	            IF ("IdbC05_Loader".M_01.startedForward OR NOT "DbDeviceONOF".boolValues[4])
	                AND ("IdbC05_Loader".M_02.startedForward OR NOT "DbDeviceONOF".boolValues[5])
	                AND (NOT "IdbC05_Loader".M_03.startedForward OR NOT "DbDeviceONOF".boolValues[6])
	                AND (NOT "IdbC05_Loader".M_04.startedForward OR NOT "DbDeviceONOF".boolValues[7])
	                OR #HMINexStep THEN
	                #HMINexStep := FALSE;
	                #StepOld := #Step;
	                #TimeCurrentStep := 0;
	                #Step := 34;

	            ELSIF #HMIStopProg THEN // Переход на сушильную продувку
	                #StepOld := #Step;
	                #TimeCurrentStep := 0;
	                #Step := 50;

	            ELSIF #HMIStop THEN // Переход на стоповый шаг
	                #HMIStop := 0;
	                #StepOld := #Step;
	                #TimeCurrentStep := 0;
	                #Step := 80;
	            END_IF;

	        34: //Сушка. Выход на заданную температуру
	            #TimeCurrentStep := #TimeCurrentStep + #cycleTime; //Подсчет времени текущей программы

	            //Передача параметров регулирования и старт горелок до момента подтверждения оператором остановки
	            "DbRegulatorsRetain".instMe[0].setpoint := "DbRegulatorsRetain".instMe[1].setpoint :=
	            "DbU1_Recipe".TemSet_2;

	            "DbRegulatorsRetain".instMe[0].hysteresys.stage_1 := "DbRegulatorsRetain".instMe[1].hysteresys.stage_1 :=
	            "DbU1_Recipe".GistHigh_2;

	            "DbRegulatorsRetain".instMe[0].hysteresys.stage_2 := "DbRegulatorsRetain".instMe[1].hysteresys.stage_2 :=
	            "DbU1_Recipe".GistLow_2;

	            #TimetUsed(START := TRUE,
	                       NUM := 4,
	                       TIM := 1800,
	                       SAMPLE_T := #cycleTime);

	            IF (#TemSet_2 - 2) <= ("IdbC03_Loader".TT7_10.value) OR #HMINexStep THEN
	                #HMINexStep := FALSE;
	                #StepOld := #Step;
	                #TimeCurrentStep := 0;
	                #Step := 35;
	                #TimetUsed(START := FALSE,
	                           NUM := 4);

	            ELSIF #HMIStopProg THEN // Переход на сушильную продувку
	                #StepOld := #Step;
	                #TimeCurrentStep := 0;
	                #Step := 50;

	            ELSIF #HMIStop THEN // Переход на стоповый шаг
	                #HMIStop := 0;
	                #StepOld := #Step;
	                #TimeCurrentStep := 0;
	                #Step := 80;
	            END_IF;

	        35: //Сушка. Отсчет заданного времени
	            #TimeCurrentStep := #TimeCurrentStep + #cycleTime; //Подсчет времени текущей программы
	            #TimeDryingRun := #TimeDryingRun + #cycleTime;

	            IF #TimeDryingRun > #TimeDryingSet OR #HMINexStep THEN
	                #HMINexStep := FALSE;
	                #StepOld := #Step;
	                #TimeCurrentStep := 0;
	                #Step := 50;

	            ELSIF #HMIStop THEN // Переход на стоповый шаг
	                #HMIStop := 0;
	                #StepOld := #Step;
	                #TimeCurrentStep := 0;
	                #Step := 80;

	            ELSIF #HMIStopProg THEN // Переход на сушильную продувку по кнопке
	                #StepOld := #Step;
	                #TimeCurrentStep := 0;
	                #Step := 50;

	          //  ELSIF #HMIStartClor THEN // Переход на Покраску по кнопке
	          //     #StepOld := #Step;
	          //      #TimeCurrentStep := 0;
	          //      #Step := 10;
	            END_IF;

	        40: //Окрасочная продувка
	            //Жалюзи Y1-2 открыты, приточный и вытяжные вентиляторы запущены, горелки работают.
	            //Условиями отключения режима являются: падение температуры до заданной в рецепте (условно +20)
	            //При выполнении условия продувка работает ещё около 3 минут и отключается.
	            #TimeCurrentStep := #TimeCurrentStep + #cycleTime; //Подсчет времени текущей программы

	            // Активация  и проверка положения клапанов  как для покраски
	            IF ("IdbC06_Loader".Y_1.activated OR NOT "DbDeviceONOF".boolValues[10])
	                AND ("IdbC06_Loader".Y_2.activated OR NOT "DbDeviceONOF".boolValues[11])
	                OR #HMINexStep THEN
	                #HMINexStep := FALSE;
	                #StepOld := #Step;
	                #Step := 41;

	            ELSIF #HMIStopProg THEN // Переход на стоповый шаг
	                #StepOld := #Step;
	                #TimeCurrentStep := 0;
	                #Step := 80;

	            ELSIF #HMIStop THEN // Переход на стоповый шаг
	                #HMIStop := 0;
	                #StepOld := #Step;
	                #TimeCurrentStep := 0;
	                #Step := 80;
	            END_IF;

	        41: // Окрасочная продувка: Активация приточных и вытяжных вентиляторов
	            #TimeCurrentStep := #TimeCurrentStep + #cycleTime; //Подсчет времени текущей программы

	            IF (("IdbC05_Loader".M_01.startedForward OR NOT "DbDeviceONOF".boolValues[4])
	                AND ("IdbC05_Loader".M_02.startedForward OR NOT "DbDeviceONOF".boolValues[5])
	                AND ("IdbC05_Loader".M_03.startedForward OR NOT "DbDeviceONOF".boolValues[6])
	                AND ("IdbC05_Loader".M_04.startedForward OR NOT "DbDeviceONOF".boolValues[7]))
	                OR #HMINexStep THEN
	                #HMINexStep := FALSE;
	                #StepOld := #Step;
	                #Step := 42;

	            ELSIF #HMIStopProg THEN // Переход на стоповый шаг
	                #StepOld := #Step;
	                #TimeCurrentStep := 0;
	                #Step := 80;

	            ELSIF #HMIStop THEN // Переход на стоповый шаг
	                #HMIStop := 0;
	                #StepOld := #Step;
	                #TimeCurrentStep := 0;
	                #Step := 80;
	            END_IF;

	        42: //Окрасочная продувка : Охлаждение до заданной температуры
	            #TimeCurrentStep := #TimeCurrentStep + #cycleTime; //Подсчет времени текущей программы
	            #TimePurgeRun := #TimePurgeRun + #cycleTime;

	            // Подсчет времени продувки и проверка температуры
	            // При достижение темературы до уставки, а так же при превышении максимального времени переход
	            IF #TimetUsed.done_arr[3] OR #TimePurgeRun >= #TimePurgSet
	                OR #HMINexStep THEN
	                #HMINexStep := FALSE;
	                #StepOld := #Step;
	                #Step := 80;

	            ELSIF #HMIStopProg THEN // Переход на стоповый шаг
	                #StepOld := #Step;
	                #TimeCurrentStep := 0;
	                #Step := 80;

	            ELSIF #HMIStop THEN // Переход на стоповый шаг
	                #HMIStop := 0;
	                #StepOld := #Step;
	                #TimeCurrentStep := 0;
	                #Step := 80;

	            ELSIF "DbU1_Recipe".TemSet_3 + 2 >= "IdbC03_Loader".TT7_10.value THEN
	                #TimetUsed(START := TRUE,
	                           NUM := 3,
	                           TIM := 180,
	                           SAMPLE_T := #cycleTime);
	            END_IF;

	        50:  // Сушильная продувка
	            #TimeCurrentStep := #TimeCurrentStep + #cycleTime; //Подсчет времени текущей программы

	            // Активация и проверка положения клапанов как для сушки
	            IF "IdbC06_Loader".Y_1.deactivated AND "IdbC06_Loader".Y_2.deactivated
	                OR #HMINexStep THEN
	                #HMINexStep := FALSE;
	                #StepOld := #Step;
	                #Step := 52;

	            ELSIF #HMIStopProg THEN // Переход на стоповый шаг
	                #StepOld := #Step;
	                #TimeCurrentStep := 0;
	                #Step := 80;

	            ELSIF #HMIStop THEN // Переход на стоповый шаг
	                #HMIStop := 0;
	                #StepOld := #Step;
	                #TimeCurrentStep := 0;
	                #Step := 80;
	            END_IF;

	        52: //Сушильная продувка. Ожидание снижения температуры.
	            #TimeCurrentStep := #TimeCurrentStep + #cycleTime; //Подсчет времени текущей программы
	            #TimePurgeRun := #TimePurgeRun + #cycleTime;

	            IF #TimetUsed.done_arr[3] OR #TimePurgeRun >= #TimePurgSet
	                OR #HMINexStep THEN
	                #HMINexStep := FALSE;
	                #StepOld := #Step;
	                #Step := 80;

	            ELSIF #HMIStopProg THEN // Переход на стоповый шаг
	                #StepOld := #Step;
	                #TimeCurrentStep := 0;
	                #Step := 80;

	            ELSIF #HMIStop THEN // Переход на стоповый шаг
	                #HMIStop := 0;
	                #StepOld := #Step;
	                #TimeCurrentStep := 0;
	                #Step := 80;

	            ELSIF "DbU1_Recipe".TemSet_3 + 2 >= "IdbC03_Loader".TT7_10.value THEN
	                #TimetUsed(START := TRUE,
	                           NUM := 3,
	                           TIM := 180,
	                           SAMPLE_T := #cycleTime);
	            END_IF;

	        80: // Штатная остановка ожидание завершение работы двигателей
	            #TimeCurrentStep := #TimeCurrentStep + #cycleTime; //Подсчет времени текущей программы

	            // Сброс параметров регулятора
	            "DbRegulatorsRetain".instMe[0].setpoint := "DbRegulatorsRetain".instMe[1].setpoint := 0.0;

	            "DbRegulatorsRetain".instMe[0].hysteresys.stage_1 := "DbRegulatorsRetain".instMe[1].hysteresys.stage_1 := 0.0;

	            "DbRegulatorsRetain".instMe[0].hysteresys.stage_2 := "DbRegulatorsRetain".instMe[1].hysteresys.stage_2 := 0.0;

	            //Проверка положения задвижек на соответствие завершающему шагу
	            IF NOT "IdbC06_Loader".Y_1.activated AND NOT "IdbC06_Loader".Y_2.activated
	                OR #HMINexStep THEN
	                #HMIStopProg := FALSE;
	                #HMINexStep := FALSE;
	                #StepOld := #Step;
	                #Step := 81;
	            END_IF;

	        81: // Штатная остановка ожидание завершение работы двигателей
	            #TimeCurrentStep := #TimeCurrentStep + #cycleTime; //Подсчет времени текущей программы

	            IF #TimeCurrentStep > 1
	                OR #HMINexStep THEN
	                #HMIStop := FALSE;
	                #HMINexStep := FALSE;
	                #StepOld := #Step;
	                #Step := 0;
	                #TimeCurrentStep := 0;
	            END_IF;

	        91: // Авария. Нажата аварийная кнопка
	            #TimeCurrentStep := #TimeCurrentStep + #cycleTime; //Подсчет времени текущей программы

	            IF #resetErrorCode  // Если нет этой аварии и нажата кнопка сброс, переходим на начальный шаг
	                AND   NOT #StorErr THEN
	                #StepOld := #Step;
	                #Step := 80;
	                #TimeCurrentStep := 0;
	            END_IF;

	        92: // Авария. Пожар
	            #TimeCurrentStep := #TimeCurrentStep + #cycleTime; //Подсчет времени текущей программы

	            IF #resetErrorCode  // Если нет этой аварии и нажата кнопка сброс, переходим на начальный шаг
	                AND NOT #FirerErr THEN
	                #StepOld := #Step;
	                #Step := 80;
	                #TimeCurrentStep := 0;
	            END_IF;

	        94: // Авария. Электропривода вентиляторов
	            #TimeCurrentStep := #TimeCurrentStep + #cycleTime; //Подсчет времени текущей программы

	            IF #resetErrorCode  // Если нет этой аварии и нажата кнопка сброс, переходим на начальный шаг
	                AND NOT #tempMotorError THEN
	                #StepOld := #Step;
	                #Step := 80;
	                #TimeCurrentStep := 0;

	            ELSIF #HMIStopProg THEN // Переход на стоповый шаг
	                #StepOld := #Step;
	                #TimeCurrentStep := 0;
	                #Step := 80;

	            ELSIF #HMIStop THEN // Переход на стоповый шаг
	                #StepOld := #Step;
	                #TimeCurrentStep := 0;
	                #Step := 80;

	            ELSIF #TimetUsed.done_arr[3] OR #TimePurgeRun >= #TimePurgSet THEN
	                #HMINexStep := FALSE;
	                #StepOld := #Step;
	                #Step := 80;

	            ELSIF "DbU1_Recipe".TemSet_3 + 2 >= "IdbC03_Loader".TT7_10.value THEN
	                #TimetUsed(START := TRUE,
	                           NUM := 3,
	                           TIM := 180,
	                           SAMPLE_T := #cycleTime);
	            END_IF;

	        95: // Авария. Высокая температура в камере.
	            #TimeCurrentStep := #TimeCurrentStep + #cycleTime; //Подсчет времени текущей программы

	            IF #resetErrorCode  // Если нет этой аварии и нажата кнопка сброс, переходим на начальный шаг
	                AND NOT #tempHiTempErr THEN
	                #StepOld := #Step;
	                #Step := 80;
	                #TimeCurrentStep := 0;

	            ELSIF #HMIStopProg THEN // Переход на стоповый шаг
	                #StepOld := #Step;
	                #TimeCurrentStep := 0;
	                #Step := 80;

	            ELSIF #HMIStop THEN // Переход на стоповый шаг
	                #StepOld := #Step;
	                #TimeCurrentStep := 0;
	                #Step := 80;

	            ELSIF #TimetUsed.done_arr[3] OR #TimePurgeRun >= #TimePurgSet THEN
	                #HMINexStep := FALSE;
	                #StepOld := #Step;
	                #Step := 80;

	            ELSIF "DbU1_Recipe".TemSet_3 + 2 >= "IdbC03_Loader".TT7_10.value THEN
	                #TimetUsed(START := TRUE,
	                           NUM := 3,
	                           TIM := 180,
	                           SAMPLE_T := #cycleTime);
	            END_IF;

	        96: // Авария. Авария оборудования.
	            #TimeCurrentStep := #TimeCurrentStep + #cycleTime; //Подсчет времени текущей программы

	            // Сброс параметров регулятора
	            "DbRegulatorsRetain".instMe[0].setpoint := "DbRegulatorsRetain".instMe[1].setpoint := 0.0;

	            "DbRegulatorsRetain".instMe[0].hysteresys.stage_1 := "DbRegulatorsRetain".instMe[1].hysteresys.stage_1 := 0.0;

	            "DbRegulatorsRetain".instMe[0].hysteresys.stage_2 := "DbRegulatorsRetain".instMe[1].hysteresys.stage_2 := 0.0;

	            IF #resetErrorCode  // Если нет этой аварии и нажата кнопка сброс, переходим на начальный шаг
	                AND NOT #tempEquipmentError THEN
	                #StepOld := #Step;
	                #Step := 80;
	                #TimeCurrentStep := 0;

	            ELSIF #HMIStopProg THEN // Переход на стоповый шаг
	                #StepOld := #Step;
	                #TimeCurrentStep := 0;
	                #Step := 80;

	            ELSIF #HMIStop THEN // Переход на стоповый шаг
	                #StepOld := #Step;
	                #TimeCurrentStep := 0;
	                #Step := 80;

	            ELSIF #TimetUsed.done_arr[3] OR #TimePurgeRun >= #TimePurgSet THEN
	                #HMINexStep := FALSE;
	                #StepOld := #Step;
	                #Step := 80;

	            ELSIF "DbU1_Recipe".TemSet_3 + 2 >= "IdbC03_Loader".TT7_10.value THEN
	                #TimetUsed(START := TRUE,
	                           NUM := 3,
	                           TIM := 180,
	                           SAMPLE_T := #cycleTime);
	            END_IF;

	        97: // Авария. Сторожевой таймер.
	            #TimeCurrentStep := #TimeCurrentStep + #cycleTime; //Подсчет времени текущей программы

	            IF #resetErrorCode  // Если нет этой аварии и нажата кнопка сброс, переходим на начальный шаг
	                AND NOT #tempWatchdogErr THEN
	                #TimeCurrentStep := 0;
	                #StepOld := #Step;
	                #Step := 80;

	            ELSIF #HMIStopProg THEN // Переход на стоповый шаг
	                #StepOld := #Step;
	                #TimeCurrentStep := 0;
	                #Step := 80;

	            ELSIF #HMIStop THEN // Переход на стоповый шаг
	                #StepOld := #Step;
	                #TimeCurrentStep := 0;
	                #Step := 80;
	            END_IF;
	    END_CASE;
	END_REGION

	REGION Активация устройств

	    CASE #Step OF

	        10, 40: // Активация начального положения задвижек. Для программы окраски
	                // задвижки Y1-2 открыты
	            IF "DbDeviceONOF".boolValues[10] THEN
	                    "IdbC06_Loader".Y_1.autoDeactivate := FALSE;
	                    "IdbC06_Loader".Y_1.autoActivate := TRUE;
	                END_IF;
	                IF "DbDeviceONOF".boolValues[11] THEN
	                    "IdbC06_Loader".Y_2.autoDeactivate := FALSE;
	                    "IdbC06_Loader".Y_2.autoActivate := TRUE;
	                END_IF;

	            11, 41: //Поочередная активация двигателей для покраски
	                //Поочередная активация двигателей
	            CASE #EM.group OF
	                #EMPTY:
	                    #EM.group := #M1_START_RELEASE;
	                    IF #TimetUsed.done_arr[1] THEN
	                        #TimetUsed(START := TRUE,
	                                   NUM := 1,
	                                   TIM := #TimeOnMotor,
	                                   SAMPLE_T := #cycleTime);
	                    END_IF;

	                    //Активация востребованности двигателей через задержку по времени
	                #M1_START_RELEASE:
	                    #TimetUsed(START := TRUE,
	                               NUM := 1,
	                               TIM := #TimeOnMotor,
	                               SAMPLE_T := #cycleTime);
	                    IF #TimetUsed.done_arr[1] THEN
	                        #EM.group := #M3_START_RELEASE;
	                        #TimetUsed(START := FALSE,
	                                   NUM := 1);
	                    END_IF;

	                #M3_START_RELEASE:
	                    #TimetUsed(START := TRUE,
	                               NUM := 1,
	                               TIM := #TimeOnMotor,
	                               SAMPLE_T := #cycleTime);
	                    IF #TimetUsed.done_arr[1] THEN
	                        #EM.group := #M2_START_RELEASE;
	                        #TimetUsed(START := FALSE,
	                                   NUM := 1);
	                    END_IF;

	                #M2_START_RELEASE:
	                    #TimetUsed(START := TRUE,
	                               NUM := 1,
	                               TIM := #TimeOnMotor,
	                               SAMPLE_T := #cycleTime);
	                    IF #TimetUsed.done_arr[1] THEN
	                        #EM.group := #M4_START_RELEASE;
	                        #TimetUsed(START := FALSE,
	                                   NUM := 1);
	                    END_IF;

	                #M4_START_RELEASE:
	                    #EM.group := #DONE;

	                #DONE:
	                    #TimetUsed(START := TRUE,
	                               NUM := 1,
	                               TIM := #TimeOnMotor,
	                               SAMPLE_T := #cycleTime);
	                    IF #TimetUsed.done_arr[1] THEN
	                        #TimetUsed(START := FALSE,
	                                   NUM := 1);
	                        #EM.group := #EMPTY;
	                    END_IF;
	                ELSE
	                    #EM.group := #EMPTY;
	                    #TimetUsed(START := FALSE,
	                               NUM := 1);
	            END_CASE;

	            // Непосредственное включение двигателей при их востребованности и разрешение (активен бит их участия в работе HMI)
	            IF ("DbDeviceONOF".boolValues[4] AND ((#EM.group >= #M1_START_RELEASE))) THEN
	                "IdbC05_Loader".M_01.autoStartForward := TRUE;
	            END_IF;
	            IF "DbDeviceONOF".boolValues[5] AND (#EM.group >= #M2_START_RELEASE) THEN
	                "IdbC05_Loader".M_02.autoStartForward := TRUE;
	            END_IF;
	            IF ("DbDeviceONOF".boolValues[6] AND (#EM.group >= #M3_START_RELEASE)) THEN
	                "IdbC05_Loader".M_03.autoStartForward := TRUE;
	            END_IF;
	            IF ("DbDeviceONOF".boolValues[7] AND (#EM.group >= #M4_START_RELEASE)) THEN
	                "IdbC05_Loader".M_04.autoStartForward := TRUE;
	            END_IF;

	        12: //Непосредственное включение двигателей и горелок для покраски.
	            //Активация горелок
	            IF "DbDeviceONOF".boolValues[8] THEN
	                "IdbC08_Loader".Regul_1.release := TRUE;
	            END_IF;
	            IF "DbDeviceONOF".boolValues[9] THEN
	                "IdbC08_Loader".Regul_2.release := TRUE;
	            END_IF;

	        30: //Переключение клапанов в режим сушки Y1-2 закрываются
	            //Активация горелок в случае деактивации. Двигатели продолжают работы до перехода на следующий шаг
	            //Деактивация горелок
	            IF "DbDeviceONOF".boolValues[8] THEN
	                "IdbC08_Loader".Regul_1.release := FALSE;
	            END_IF;
	            IF "DbDeviceONOF".boolValues[9] THEN
	                "IdbC08_Loader".Regul_2.release := FALSE;
	            END_IF;

	            // Деактивация двигателей
	            "IdbC05_Loader".M_01.autoStartForward := "IdbC05_Loader".M_02.autoStartForward := "IdbC05_Loader".M_03.autoStartForward := "IdbC05_Loader".M_04.autoStartForward := FALSE;

	            //Переключение клапанов в режим сушки
	            IF "DbDeviceONOF".boolValues[10] THEN
	                "IdbC06_Loader".Y_1.autoActivate := FALSE;
	                "IdbC06_Loader".Y_1.autoDeactivate := TRUE;
	            END_IF;
	            IF "DbDeviceONOF".boolValues[11] THEN
	                "IdbC06_Loader".Y_2.autoActivate := FALSE;
	                "IdbC06_Loader".Y_2.autoDeactivate := TRUE;
	            END_IF;

	        32:  // Поочередное включение двигателей
	                CASE #EM.group OF
	                    #EMPTY:
	                        #EM.group := #M1_START_RELEASE;
	                        IF #TimetUsed.done_arr[1] THEN
	                            #TimetUsed(START := TRUE,
	                                       NUM := 1,
	                                       TIM := #TimeOnMotor,
	                                       SAMPLE_T := #cycleTime);
	                        END_IF;

	                        //Активация востребованности двигателей через задержку по времени
	                    #M1_START_RELEASE:
	                        #TimetUsed(START := TRUE,
	                                   NUM := 1,
	                                   TIM := #TimeOnMotor,
	                                   SAMPLE_T := #cycleTime);
	                        IF #TimetUsed.done_arr[1] THEN
	                            #EM.group := #M2_START_RELEASE;
	                            #TimetUsed(START := FALSE,
	                                       NUM := 1);
	                        END_IF;

	                    #M2_START_RELEASE:
	                        #EM.group := #DONE;

	                    #DONE:
	                        #TimetUsed(START := TRUE,
	                                   NUM := 1,
	                                   TIM := #TimeOnMotor,
	                                   SAMPLE_T := #cycleTime);
	                        IF #TimetUsed.done_arr[1] THEN
	                            #EM.group := #EMPTY;
	                            #TimetUsed(START := FALSE,
	                                       NUM := 1);
	                        END_IF;
	                    ELSE
	                        #EM.group := #EMPTY;
	                        #TimetUsed(START := FALSE,
	                                   NUM := 1);
	                END_CASE;

	                // Непосредственное включение двигателей при их востребованности и разрешение (активен бит их участия в работе HMI)
	                IF ("DbDeviceONOF".boolValues[4] AND ((#EM.group >= #M1_START_RELEASE))) THEN
	                    "IdbC05_Loader".M_01.autoStartForward := TRUE;
	                END_IF;
	                IF "DbDeviceONOF".boolValues[5] AND (#EM.group >= #M2_START_RELEASE) THEN
	                    "IdbC05_Loader".M_02.autoStartForward := TRUE;
	                END_IF;
	                IF "DbDeviceONOF".boolValues[6] THEN
	                    "IdbC05_Loader".M_03.autoStartForward := FALSE;
	                END_IF;
	                IF "DbDeviceONOF".boolValues[7] THEN
	                    "IdbC05_Loader".M_04.autoStartForward := FALSE;
	                END_IF;

	        34: // Активация горелок
	            IF "DbDeviceONOF".boolValues[8] THEN
	                "IdbC08_Loader".Regul_1.release := TRUE;
	            END_IF;
	            IF "DbDeviceONOF".boolValues[9] THEN
	                "IdbC08_Loader".Regul_2.release := TRUE;
	            END_IF;

	        42: //Окрасочная продувка. Ожидание достижения уставок по времени или температуре
	            //Деактивация горелок
	            IF "DbDeviceONOF".boolValues[8] THEN
	                "IdbC08_Loader".Regul_1.release := FALSE;
	            END_IF;
	            IF "DbDeviceONOF".boolValues[9] THEN
	                "IdbC08_Loader".Regul_2.release := FALSE;
	            END_IF;

	        50: //Сушильная продувка
	            //Клапаны в режиме сушки, остаются в предыдущем положении
	            IF "DbDeviceONOF".boolValues[10] THEN
	                "IdbC06_Loader".Y_1.autoActivate := FALSE;
	                "IdbC06_Loader".Y_1.autoDeactivate := TRUE;
	            END_IF;
	            IF "DbDeviceONOF".boolValues[11] THEN
	                "IdbC06_Loader".Y_2.autoActivate := FALSE;
	                "IdbC06_Loader".Y_2.autoDeactivate := TRUE;
	            END_IF;

	        52: //Сушильная продувка
	            // Приточне двигатели продолжают работу, вытяжные деактивированы.
	            IF ("DbDeviceONOF".boolValues[4]) THEN
	                "IdbC05_Loader".M_01.autoStartForward := TRUE;
	            END_IF;
	            IF "DbDeviceONOF".boolValues[5] THEN
	                "IdbC05_Loader".M_02.autoStartForward := TRUE;
	            END_IF;
	            IF ("DbDeviceONOF".boolValues[6]) THEN
	                "IdbC05_Loader".M_03.autoStartForward := FALSE;
	            END_IF;
	            IF ("DbDeviceONOF".boolValues[7]) THEN
	                "IdbC05_Loader".M_04.autoStartForward := FALSE;
	            END_IF;

	            // Деактивация регулирования горелок
	            "IdbC08_Loader".Regul_1.release := FALSE;
	            "IdbC08_Loader".Regul_2.release := FALSE;

	        80:  //Переключенеи задвижек в первоначальное положение, дективация остального
	            // задвижек жалюзи Y1-2 закрыты
	            IF "DbDeviceONOF".boolValues[10] THEN
	                "IdbC06_Loader".Y_1.autoActivate := FALSE;
	                "IdbC06_Loader".Y_1.autoDeactivate := TRUE;
	            END_IF;
	            IF "DbDeviceONOF".boolValues[11] THEN
	                "IdbC06_Loader".Y_2.autoActivate := FALSE;
	                "IdbC06_Loader".Y_2.autoDeactivate := TRUE;
	            END_IF;

	            // Деактивация горелок
	            "IdbC08_Loader".Regul_1.release := FALSE;
	            "IdbC08_Loader".Regul_2.release := FALSE;

	            // Деактивация двигателей
	            "IdbC05_Loader".M_01.autoStartForward := "IdbC05_Loader".M_02.autoStartForward := "IdbC05_Loader".M_03.autoStartForward := "IdbC05_Loader".M_04.autoStartForward := FALSE;

	        81: // Деактивация всего
	            //Переключение камер задвижек 1-2
	            "IdbC06_Loader".Y_1.autoActivate := "IdbC06_Loader".Y_2.autoActivate := FALSE;
	            "IdbC06_Loader".Y_1.autoDeactivate := "IdbC06_Loader".Y_2.autoDeactivate := TRUE;

	            // Деактивация горелок
	            "IdbC08_Loader".Regul_1.release := FALSE;
	            "IdbC08_Loader".Regul_2.release := FALSE;

	            // Деактивация двигателей
	            "IdbC05_Loader".M_01.autoStartForward := "IdbC05_Loader".M_02.autoStartForward := "IdbC05_Loader".M_03.autoStartForward := "IdbC05_Loader".M_04.autoStartForward := FALSE;

	        91: //Нажата аварийная кнопка. Все отключить
	            // Аварийный останов активируетя до перехода на шаг
	            //Отключение в авто режиме
	            //Отключение   задвижек 1-2
	            "IdbC06_Loader".Y_1.autoActivate := "IdbC06_Loader".Y_2.autoActivate := FALSE;
	            "IdbC06_Loader".Y_1.autoDeactivate := "IdbC06_Loader".Y_2.autoDeactivate := TRUE;

	            // Деактивация горелок
	            "IdbC08_Loader".Regul_1.release := FALSE;
	            "IdbC08_Loader".Regul_2.release := FALSE;

	            // Деактивация двигателей
	            "IdbC05_Loader".M_01.autoStartForward := "IdbC05_Loader".M_02.autoStartForward := "IdbC05_Loader".M_03.autoStartForward := "IdbC05_Loader".M_04.autoStartForward := FALSE;

	        92: // Сигнал о пожаре. Y1-2 закрываются, свет горит на протяжении 30 секунд и отключается.
	            // Аварийный останов активируетя до перехода на шаг
	            //Отключение в авто режиме

	            //Переключение клапанов в режим сушки
	            IF "DbDeviceONOF".boolValues[10] THEN
	                "IdbC06_Loader".Y_1.autoActivate := FALSE;
	                "IdbC06_Loader".Y_1.autoDeactivate := TRUE;
	            END_IF;
	            IF "DbDeviceONOF".boolValues[11] THEN
	                "IdbC06_Loader".Y_2.autoActivate := FALSE;
	                "IdbC06_Loader".Y_2.autoDeactivate := TRUE;
	            END_IF;

	            "IdbC08_Loader".Regul_1.release := FALSE;
	            "IdbC08_Loader".Regul_2.release := FALSE;

	            // Деактивация двигателей
	            "IdbC05_Loader".M_01.autoStartForward := "IdbC05_Loader".M_02.autoStartForward := "IdbC05_Loader".M_03.autoStartForward := "IdbC05_Loader".M_04.autoStartForward := FALSE;

	        94: // Авария привода вентилятора
	            //Запускается режим продувки. Тип продувки зависит от того на какой из программ это произошло.
	            // Задвижки остаются в предыдущем положении

	            //Горелки останавливаются
	            "IdbC08_Loader".Regul_1.release := FALSE;
	            "IdbC08_Loader".Regul_2.release := FALSE;

	            // Активируются только приточка Если какой-то в аварии он и так не запустится
	            IF (#StepOld >= 30 AND #StepOld < 40) OR (#StepOld >= 50 AND #StepOld < 60) THEN // Если пред шаг связан с сушкой, то запускается сушильная продувка
	                "IdbC05_Loader".M_01.autoStartForward := "IdbC05_Loader".M_02.autoStartForward := TRUE;
	                "IdbC05_Loader".M_03.autoStartForward := "IdbC05_Loader".M_04.autoStartForward := FALSE;
	            ELSE // Иначе запускается продувка с работой всех двигателей
	                "IdbC05_Loader".M_01.autoStartForward := "IdbC05_Loader".M_02.autoStartForward := "IdbC05_Loader".M_03.autoStartForward := "IdbC05_Loader".M_04.autoStartForward := TRUE;
	            END_IF;

	        95, 96: // Авария  оборудования или Высокая температура в камере.
	            //Запускается режим продувки. Тип продувки зависит от того на какой из программ это произошло.
	            // Задвижки остаются в предыдущем положении
	            //Горелки останавливаются
	            "IdbC08_Loader".Regul_1.release := FALSE;
	            "IdbC08_Loader".Regul_2.release := FALSE;

	            // Активируются все двигатели. Если какой-то в аварии он и так не запустится
	            IF (#StepOld >= 30 AND #StepOld < 40) OR (#StepOld >= 50 AND #StepOld < 60) THEN // Если пред шаг связан с сушкой, то запускается сушильная продувка
	                "IdbC05_Loader".M_01.autoStartForward := "IdbC05_Loader".M_02.autoStartForward := TRUE;
	                "IdbC05_Loader".M_03.autoStartForward := "IdbC05_Loader".M_04.autoStartForward := FALSE;
	            ELSE // Иначе запускается продувка с работой всех двигателей
	                "IdbC05_Loader".M_01.autoStartForward := "IdbC05_Loader".M_02.autoStartForward := "IdbC05_Loader".M_03.autoStartForward := "IdbC05_Loader".M_04.autoStartForward := TRUE;
	            END_IF;

	        97: //Активирован сторожевой таймер. Все отключить
	            "IdbC06_Loader".Y_1.autoActivate := "IdbC06_Loader".Y_2.autoActivate := FALSE;
	            "IdbC06_Loader".Y_1.autoDeactivate := "IdbC06_Loader".Y_2.autoDeactivate := TRUE;

	            // Деактивация горелок
	            "IdbC08_Loader".Regul_1.release := FALSE;
	            "IdbC08_Loader".Regul_2.release := FALSE;

	            // Деактивация двигателей
	            "IdbC05_Loader".M_01.autoStartForward := "IdbC05_Loader".M_02.autoStartForward := "IdbC05_Loader".M_03.autoStartForward := "IdbC05_Loader".M_04.autoStartForward := FALSE;
	    END_CASE;
	END_REGION

	REGION Активация освещения
	    //Активация свет 1 во время работы
	    IF ((#Step >  0 AND #Step <= 13)  // Работа во время основной программы
	        OR (#Step = 92 AND #TimeCurrentStep <30)//Работа во время аварии по пожару
	        OR ("HL_01_ManOn" AND NOT #StorErr))
	        AND "DbDeviceONOF".boolValues[12] THEN// Свет
	        "IdbC02_Loader".HL_01.release := TRUE;
	    ELSE
	        "IdbC02_Loader".HL_01.release  := FALSE;
	    END_IF;
	END_REGION

	REGION Сброс
	    #HMITime := UDINT_TO_TOD(REAL_TO_UDINT(#TimeCurrentStep * 1000.0));
	    #HMITimeAll := UDINT_TO_TOD(REAL_TO_UDINT(#TimeRunAll * 1000.0));

	    #tempError := #hmiErrorConfirm <> w#16#0;
	    #tempWarning := #hmiWarningConfirm <> w#16#0;

	    #hmiControl_1 := w#16#0; //Сброс контрольного слова

	    IF #tempHmiResetErrorCode THEN // Сброс аварий
	        #hmiErrorConfirm := w#16#0;
	        #tempHmiResetErrorCode := FALSE;
	        #resetErrorCode := TRUE;
	    ELSE
	        #resetErrorCode := FALSE ;
	    END_IF;

	    IF #tempHmiResetWarningCode THEN // Сброс предупреждений
	        #hmiWarningConfirm := w#16#0;
	        #tempHmiResetWarningCode := FALSE;
	    END_IF;

	    // Сброс нажатий с панели
	    #HMIStop := False;
	    #HMINexStep := False;
	    #HMIStartClor := FALSE;
	    #HMIStartDrying := FALSE;
	    #HMIStopProg := FALSE;
	END_REGION
END_FUNCTION_BLOCK

